{attribute 'qualified_only'}
{attribute 'to_string'}
TYPE E_KNXnetIP_ServiceTypes :
(
	eL_DataReq		 	:= 16#11,
	eL_DataCon			:= 16#2E,
	eL_DataInd			:= 16#29
)BYTE
;
END_TYPE

(* stored: Version 1.1.0.1
   DUT E_KNXnetIP_ServiceTypes: Id {0bd02cdd-29b4-4240-bc39-365917793720} *)
